# B&R Automation Studio project DataflowProgramming
Automation Studio 4.7.2.98

## Configuration _STD

CPU X20cCP1586, AutomationRuntime C4.72, Build 6.3.0, Vc V4.15.4

### Task classes (Cpu.sw)
```
Cyclic#4:
  Dataflow <- _dataflow.Dataflow.prg
  DataflowMi <- _dataflow.DataflowMirror.prg
```

### Hardware
```
X20cCP1586 : X20cCP1586 v1.6.0.0
  Connector IF2:
    ActivateDevice = 1
  ConfigurationID = DataflowProgramming__STD
  Simulation = 1
```

## Logical view

Binary libraries used (declarations not repeated): operator, runtime, astime, AsIecCon

### Global.typ - Global data types
```iecst
(********************************************************************
 * COPYRIGHT --
 ********************************************************************
 * File: Global.typ
 * Author: k1008014
 * Created: July 13, 2020
 ********************************************************************
 * Global data types of project DataflowProgramming
 ********************************************************************)

TYPE
	DataFlow : 	STRUCT
		O_Out : BOOL;
		I_In : BOOL;
		I_Enable : BOOL;
	END_STRUCT;
END_TYPE
```

### Package Logical/Libraries - Global libraries

### Variables.var - Local variables
```iecst
VAR
	test : DataFlow;
END_VAR
```

### Program Logical/_dataflow/Dataflow (ANSIC)

#### Dataflow.cpp - Implementation code
```cpp
/********************************************************************
 * COPYRIGHT --
 ********************************************************************
 * Program: Dataflow
 * File: Dataflow.cpp
 * Author: k1008014
 * Created: July 13, 2020
 ********************************************************************
 * Implementation of program Dataflow
 ********************************************************************/

#ifdef _SG4 /*IF B&R system*/ //TODO -> Add where needed
#include <bur/plctypes.h>
#include "plcdeclarations.h"
#ifdef _DEFAULT_INCLUDES
	#include <AsDefault.h>
#endif
#endif

#include "generaldefines.h"
#include "Manager.hpp"

unsigned long bur_heap_size=0xFFFFF;

dataflow::Manager* t_man;
extern DataFlow test;
dataflow::INode* ptr;
bool _trigflag;

#define _TEST_NODE_A 0
#define _TEST_NODE_B 1
#define _TEST_NODE_C 2

void ManagerSetup()
{
	/*Prepare manager*/
	t_man->ClearManager();
	t_man->AddNode(new dataflow::NOT()); // _TEST_NODE_A
	t_man->AddNode(new dataflow::NOT()); // _TEST_NODE_B
	t_man->AddNode(new dataflow::NOT()); // _TEST_NODE_C
	t_man->InitExecution();
	/*Set nodes links*/
	/***********************************************/
	/***********************************************/
//_TEST_NODE_A
	ptr = t_man->GetNodePtr(_TEST_NODE_A);
	ptr->SetInput(&test.I_In,0);
	//ptr->SetOutput(&test.O_Out,0); //Forcing output to a different location
	/***********************************************/
	/***********************************************/
//_TEST_NODE_B
	ptr = t_man->GetNodePtr(_TEST_NODE_B);
	/*Output is created with node init
	 *when an output channel is created its memory is allocated for the type declared
	 */
	ptr->SetInput(t_man->GetNodePtr(_TEST_NODE_A)->GetOutputPtr(0),0);
	//ptr->SetOutput(&test.O_Out,0); //Forcing output to a different location
//_TEST_NODE_C
	ptr = t_man->GetNodePtr(_TEST_NODE_C);
	/*Output is created with node init
	 *when an output channel is created its memory is allocated for the type declared
	 */
	ptr->SetInput(t_man->GetNodePtr(_TEST_NODE_B)->GetOutputPtr(0),0);
	ptr->SetOutput(&test.O_Out,0); //Forcing output to a different location
}

void _INIT DataflowInit(void)
{
	t_man = new dataflow::Manager();
	ManagerSetup();
}

void _CYCLIC DataflowCyclic(void)
{
	/*Manager cyclic*/
	if(test.I_In && (_trigflag != test.I_In))
	{
		ManagerSetup();
	}
	/*R_TRIG*/
	_trigflag = test.I_In;

	/*Adds control to execution, only for test purposes*/
	if(test.I_Enable)
	{
		t_man->CyclicExecution();
	}
	test.O_Out = test.O_Out;
}
```

#### plcdeclarations.h
```c
/********************************************************************
 * COPYRIGHT --
 ********************************************************************
 * Program: Dataflow
 * File: PlcDeclarations.h
 * Author: k1008014
 * Created: July 13, 2020
 *******************************************************************/

#include <bur/plctypes.h>
```

#### plcdeclarations.c
```c
#include <bur/plctypes.h>

#ifdef _DEFAULT_INCLUDES
	#include <AsDefault.h>
#endif

/*Varible definitions*/
_GLOBAL BOOL isTrue;
```

#### generaldefines.h
```c
/********************************************************************
 * COPYRIGHT --
 ********************************************************************
 * Program: Dataflow
 * File: GeneralDefines.h
 * Author: k1008014
 * Created: July 13, 2020
 *******************************************************************/

#ifndef GENERAL_DEFINES_H
#define GENERAL_DEFINES_H

//#define _DATAFLOW_LOGGER

#include <bur/plctypes.h>

namespace dataflow
{

	enum _types { _INT, _DOUBLE, _FLOAT, _CHAR, _STRING, _REAL, _BOOL };
	enum _fubs  { _LT, _GT, _AND, _OR, _OUT, _CONST, _VAR };

}

#endif
```

#### INode.hpp
```cpp
/********************************************************************
 * COPYRIGHT --
 ********************************************************************
 * Program: Dataflow
 * File: INode.hpp
 * Author: k1008014
 * Created: July 13, 2020
 *******************************************************************/

#ifndef NODE_HPP
#define NODE_HPP

#include <bur/plctypes.h>
#include <vector>

#include "Input_channel.hpp"
#include "Output_channel.hpp"

namespace dataflow
{
	class NodeException: public std::exception
	{
		virtual const char* what() const throw()
		{
			return "Node exception";
		}
	} NodeEx;

	class INode
	{
		public:

		plcbit error;

		/// <summary>Add an input to the node</summary>
		/// <param name="type">Specifies the type of the input</param>
		/// <returns>void</returns>
		void AddInput(int type)
		{
			try
			{
				this->inputs.push_back(new Input_channel(type));
			}
			catch(std::bad_alloc& e)
			{
				this->error = 1;
			}
		}

		/// <summary>Set pointer to an input linking the node to an ouput or val</summary>
		/// <param name="ptr">void* to another node or value, user must check types</param>
		/// <param name="inputNr">Input number to set, if out of bound throw NodeEx</param>
		/// <returns>void</returns>
		void SetInput(void* ptr, int inputNr)
		{
			if(((this->inputs.size() + 1) < inputNr) || inputNr < 0)
			{
				throw NodeEx;
			}
			this->inputs[inputNr]->setPointer(ptr);
		}

		/// <summary>Set pointer to an output linking the node to an input or val</summary>
		/// <param name="ptr">void* to another node or value, user must check types</param>
		/// <param name="inputNr">Output number to set, if out of bound throw NodeEx</param>
		/// <returns>void</returns>
		void SetOutput(void* ptr, int outPutNr)
		{
			if(((this->outputs.size() + 1) < outPutNr) || outPutNr < 0)
			{
				this->error = 1;
				throw NodeEx;
			}
			this->outputs[outPutNr]->setPointer((void*)ptr);
		}

		/// <summary>Add an output to the node</summary>
		/// <param name="type">Specifies the type of the output</param>
		/// <returns>void</returns>
		void AddOutput(int type)
		{
			try
			{
				this->outputs.push_back(new Output_channel(type));
			}
			catch(std::bad_alloc& e)
			{
				this->error = 1;
			}
		}

		/// <summary>Get ouput pointer</summary>
		/// <param name="type">Specifies the output number</param>
		/// <returns>void*</returns>
		void* GetOutputPtr(int outPutNr)
		{
			if(((this->outputs.size() + 1) < outPutNr) || outPutNr < 0)
			{
				this->error = 1;
				throw NodeEx;
			}
			else
			{
				return this->outputs[outPutNr]->getPointer();
			}
		}

		/// <summary>Virtual method, Init node</summary>
		/// <returns>void</returns>
		virtual void Init() = 0;
		/// <summary>Virtual method, Cyclic executon of the node[main logic]</summary>
		/// <returns>void</returns>
		virtual void Cyclic() = 0;
		/// <summary>Virtual method, Exit function on decostruction</summary>
		/// <returns>void</returns>
		virtual void Exit() = 0;

		protected:
		/*Vectors of I/O*/
		std::vector<Input_channel*> inputs;
		std::vector<Output_channel*> outputs;

	};
}

#endif
```

#### Input_channel.hpp
```cpp
/********************************************************************
 * COPYRIGHT --
 ********************************************************************
 * Program: Dataflow
 * File: Input_channel.hpp
 * Author: k1008014
 * Created: July 13, 2020
 *******************************************************************/

/*Include guards*/
#ifndef INPUT_CHANNEL_HPP
#define INPUT_CHANNEL_HPP

#include <bur/plctypes.h>
#include "generaldefines.h"

/*Template class for every type in input*/
class Input_channel {

	void* value;
	int Type;

	public:

	Input_channel(int type)
	{
		this->Type = type;
		/*Alloc internal memory for the value*/
		CastDynamicType();
	}
	//Return type name of the input demangled
	//[typeid return from type_info is compiler dependant and needs to be demangled]
	int getType()
	{
		/*std::type_info  &ti = typeid(this->value);
		return abi::__cxa_demangle(ti.name(), 0, 0, 0);*/
		return this->Type;
	}
	//Return value
	void* getVal()
	{
		return value;
	}

	//Return pointer to value
	void* getPointer()
	{
		return &this->value;
	}

	void setPointer(void* ptr)
	{
		this->value = (void*)ptr;
	}

	//Type must be defined at alloc time
	//Cast the input void* to type*
	//TODO -> erase this, has no sense
	void CastDynamicType()
	{
		switch (this->Type)
		{
			case dataflow::_INT:
				static_cast<int*>(value);
				break;
			case dataflow::_FLOAT:
				static_cast<float*>(value);
				break;
			case dataflow::_CHAR:
				static_cast<char*>(value);
				break;
			case dataflow::_DOUBLE:
				static_cast<double*>(value);
				break;
			case dataflow::_BOOL:
				static_cast<plcbit*>(value);
				break;
			default:
				break;
		}
	}
};

#endif
```

#### Output_channel.hpp
```cpp
/********************************************************************
 * COPYRIGHT --
 ********************************************************************
 * Program: Dataflow
 * File: Output_channel.hpp
 * Author: k1008014
 * Created: July 13, 2020
 *******************************************************************/

#ifndef OUTPUT_CHANNEL_HPP
#define OUTPUT_CHANNEL_HPP

#include <bur/plctypes.h>
#include "generaldefines.h"
#include <cstdlib>

/*Template class for every type in output*/
class Output_channel {

	void* value;
	int Type;

	public:

	Output_channel(int type)
	{
		this->Type = type;
		/*Alloc internal memory for the value*/
		AllocDynamicOutput();
	}
	//Return type name of the input demangled
	//[typeid return from type_info is compiler dependant and needs to be demangled]
	int getType()
	{
		/*std::type_info  &ti = typeid(this->value);
		return abi::__cxa_demangle(ti.name(), 0, 0, 0);*/
		return this->Type;
	}
	//Return value
	void* getVal()
	{
		return value;
	}
	//Return pointer to value
	void* getPointer()
	{
		return this->value;
	}

	void setPointer(void* ptr)
	{
		this->value = ptr;
	}

	//Type must be defined at alloc time
	//alloc memory in order to get space into memory for the type
	//and then cast the void* to type*
	void AllocDynamicOutput()
	{
		switch (this->Type)
		{
			case dataflow::_INT:
				value = malloc(sizeof(int));
				static_cast<int*>(value);
				break;
			case dataflow::_FLOAT:
				value = malloc(sizeof(float));
				static_cast<float*>(value);
				break;
			case dataflow::_CHAR:
				value = malloc(sizeof(char));
				static_cast<char*>(value);
				break;
			case dataflow::_DOUBLE:
				value = malloc(sizeof(double));
				static_cast<double*>(value);
				break;
			case dataflow::_BOOL:
				value = malloc(sizeof(plcbit));
				static_cast<plcbit*>(value);
				break;
			default:
				break;
		}
	}
};

#endif
```

#### NodeFunctions.hpp
```cpp
/********************************************************************
 * COPYRIGHT --
 ********************************************************************
 * Program: Dataflow
 * File: NodeFunctions.hpp
 * Author: k1008014
 * Created: July 13, 2020
 *******************************************************************/
#ifndef NODE_GENERAL_FUNCTIONS_HPP
#define NODE_GENERAL_FUNCTIONS_HPP

#include <bur/plctypes.h>
#include "INode.hpp"

namespace dataflow
{

	/*Less then*/
	class LT: public INode
	{
		private:

		bool outVal;

		public:

		/// <summary>Init node, set standard structure</summary>
		/// <returns>void</returns>
		void Init()
		{
			//Input 1
			this->AddInput(dataflow::_DOUBLE);
			//Input 2
			this->AddInput(dataflow::_DOUBLE);
			//Output 1
			this->AddOutput(dataflow::_BOOL);
		}
		/// <summary>Cyclic executon of the node[main logic]</summary>
		/// <returns>void</returns>
		void Cyclic()
		{
			this->outVal = (double*)this->inputs[0]->getVal() < (double*)this->inputs[1]->getVal();
			this->SetOutput((void*)outVal,0);
		}
		/// <summary>Exit function on decostruction</summary>
		/// <returns>void</returns>
		void Exit()
		{
			return;
		}

	};
	/*Greater then*/
	class GT : public INode
	{
		private:

		bool outVal;

		public:

		/// <summary>Init node, set standard structure</summary>
		/// <returns>void</returns>
		void Init()
		{
			//Input 1
			this->AddInput(dataflow::_DOUBLE);
			//Input 2
			this->AddInput(dataflow::_DOUBLE);
			//Output 1
			this->AddOutput(dataflow::_BOOL);
		}
		/// <summary>Cyclic executon of the node[main logic]</summary>
		/// <returns>void</returns>
		void Cyclic()
		{
			this->outVal = (double*)this->inputs[0]->getVal() > (double*)this->inputs[1]->getVal();
			this->SetOutput((void*)outVal,0);
		}
		/// <summary>Exit function on decostruction</summary>
		/// <returns>void</returns>
		void Exit()
		{
			return;
		}

	};

	class VAR : public INode
	{
		public:
		/// <summary>Init node, set standard structure</summary>
		/// <returns>void</returns>
		void Init()
		{
			/*Input 1*/
			this->AddInput(dataflow::_DOUBLE);
			/*Output 1*/
			this->AddOutput(dataflow::_DOUBLE);
			/*Set bridge input-output*/
			this->SetOutput((double*)this->inputs[0]->getVal(),0);

		}

		void Cyclic()
		{
			return;
		}

		void Exit()
		{
			return;
		}
	};

	#define _1_INPUT 0
	#define _2_INPUT 1

	#define _1_OUTPUT 0
	#define _2_OUTPUT 1

	//NOT bool function
	//Now is used as test
	class NOT : public INode
	{

		private:

		plcbit outVal;

		public:

		/// <summary>Init node, set standard structure</summary>
		/// <returns>void</returns>
		void Init()
		{
			/*Input 1*/
			this->AddInput(dataflow::_BOOL);
			/*Output 1*/
			this->AddOutput(dataflow::_BOOL);
		}

		void Cyclic()
		{
			if(!this->error)
			{
				/*Static cast of input void pointer*/
				auto tmp_in = static_cast<plcbit*>(this->inputs[_1_INPUT]->getVal());
				/*Static cast of output void pointer*/
				auto tmp_out = static_cast<plcbit*>(this->GetOutputPtr(_1_OUTPUT));
				if(*tmp_in)
				{
					*tmp_out = false;
				}
				else
				{
					*tmp_out = true;
				}
			}
		}

		void Exit()
		{
			return;
		}
	};
}

#endif
```

#### Manager.hpp
```cpp
/********************************************************************
 * COPYRIGHT --
 ********************************************************************
 * Program: Dataflow
 * File: Manager.hpp
 * Author: k1008014
 * Created: July 13, 2020
 *******************************************************************/

#ifndef MANAGER_HPP
#define MANAGER_HPP

#include <bur/plctypes.h>
#include <vector>
#include <algorithm>
#include <iostream>
#include "NodeFunctions.hpp"
#include "generaldefines.h"

#ifdef _SG4 /*B&R system*/

#define _NODES_LIMITER
#define _MAX_NODES_NR 100

#endif

namespace dataflow
{

	class ManagerException: public std::exception
	{
		virtual const char* what() const throw()
		{
			return "Manager exception";
		}
	} ManagerEx;

#ifdef _NODES_LIMITER

	class ManagerNodesNumberOutOfBounds: public std::exception
	{
		virtual const char* what() const throw()
		{
		return "Manager exception : too many nodes";
		}
	} ManagerOutOfBoundEx;

#endif

	//support for foreach
	void NodeExecution(INode *node)
	{
		node->Cyclic();
	}

	//support for foreach
	void NodeInit(INode *node)
	{
		node->Init();
	}

	class Manager
	{
		private:

		std::vector<INode *> nodes;

		public:

		bool ErrorState;

		/// <summary>Get Node pointer</summary>
		/// <param name="nodeNr">Specifies the node number</param>
		/// <returns>INode*</returns>
		INode* GetNodePtr(int nodeNr)
		{
			if(((this->nodes.size() + 1) < nodeNr) || nodeNr < 0)
			{
				this->ErrorState = true;
				throw ManagerEx;
			}
			else
			{
				return this->nodes[nodeNr];
			}
		}

		/// <summary>Remove Node from manager returning a pointer of the element</summary>
		/// <param name="nodeNr">Specifies the node number</param>
		/// <returns>INode*</returns>
		INode*  RemoveNode(int nodeNr)
		{
			if(((this->nodes.size() + 1) < nodeNr) || nodeNr < 0)
			{
				this->ErrorState = true;
				throw ManagerEx;
			}
			else
			{
				auto tmp = this->nodes[nodeNr];
				this->nodes.erase(this->nodes.begin() + nodeNr);
			}
		}

		/// <summary>Exec Cyclic of every node contained into manager</summary>
		/// <returns>void</returns>
		void CyclicExecution()
		{
			std::for_each(nodes.begin(), nodes.end(), NodeExecution);
		}

		/// <summary>Exec Init of every node contained into manager</summary>
		/// <returns>void</returns>
		void InitExecution()
		{
			std::for_each(nodes.begin(), nodes.end(), NodeInit);
		}

		/*Selection of type of node*/
		static INode *SelectINode(int INodeNr)
		{
			switch (INodeNr)
			{
				case dataflow::_LT :
					return new LT();
					break;
				case dataflow::_GT :
					return new GT();
					break;
				default:
					break;
			}
		}

		/// <summary>Get Node pointer</summary>
		/// <param name="nodeNr">Specifies the node number</param>
		/// <returns>INode*</returns>
		INode **AddNode(INode *node)
		{
/*Max amount of nodes, prevent memory errors*/
#ifdef _NODES_LIMITER
			if(this->nodes.size() > _MAX_NODES_NR)
			{
				this->ErrorState = true;
				throw ManagerOutOfBoundEx;
			}
#endif
			try
			{
				this->nodes.push_back(node);
				return &node;
			}
			catch (std::exception ex)
			{
				this->ErrorState = true;
#ifdef _DATAFLOW_LOGGER
				/*TODO -> add logger*/
#endif
			}
		}

		/// <summary>Returns last node added to the manager</summary>
		/// <returns>INode*</returns>
		INode* GetLastNode()
		{
			return this->nodes.back();
		}

		/// <summary>Clear Manager memory</summary>
		/// <returns>void</returns>
		void ClearManager()
		{
			if(!this->nodes.empty())
			{
				try
				{
					this->nodes.clear();
				}
				catch (std::exception ex)
				{
					this->ErrorState = true;
#ifdef _DATAFLOW_LOGGER
					/*TODO -> add logger*/
#endif
				}
			}
		}
	};

}

#endif
```

### Program Logical/_dataflow/DataflowMirror (ANSIC)

#### Main.c - Init, cyclic, exit code
```c
#include <bur/plctypes.h>

#ifdef _DEFAULT_INCLUDES
	#include <AsDefault.h>
#endif

extern DataFlow test;

void _INIT ProgramInit(void)
{

}

void _CYCLIC ProgramCyclic(void)
{

}

void _EXIT ProgramExit(void)
{
	test.O_Out = 1;
}
```
